FUNCTION F_DegPerSecToUpm : LREAL
VAR_INPUT
	fValue : LREAL; // °/s value
END_VAR
VAR
END_VAR

F_DegPerSecToUpm := fValue * 1/6; // °/s => 1/min (x * 60/360)

END_FUNCTION

(* stored: Version 1.1.0.1, ProductVersion 3.1.4024.12
   POU F_DegPerSecToUpm: Id {f12718ca-1565-4248-b8b7-d661d1f88e56}, SpecialFunc None *)
